TYPE ST_LeakTestRecipe :
STRUCT
	nValveMask	: LWORD;
	tOnDelay	: TIME;
	tOffDelay	: TIME;
	
END_STRUCT
END_TYPE

(* stored: Version 1.1.0.1
   DUT ST_LeakTestRecipe: Id {bfb3fff6-e231-01c6-0363-151402f9c543} *)
